FUNCTION_BLOCK FB_IdleState IMPLEMENTS I_State
VAR_INPUT
END_VAR
VAR_OUTPUT
END_VAR
VAR
	pMachine : POINTER TO FB_StateMachine;
END_VAR

{warning 'Eigenschaftenimplementierung hinzufügen'}
PROPERTY Description : STRING
GET
Description := 'Heat pump is idle';
END_GET
END_PROPERTY

METHOD ErrorDetected : BOOL
VAR_INPUT
	errorEvents		: ST_ErrorEvents;
END_VAR
VAR
	message				: STRING(255);
END_VAR
message := toErrorText(errorEvents);
ADSLOGSTR(ADSLOG_MSGTYPE_HINT, 'Error detected -> Error:  %s', message);
pMachine^.SetState(pMachine^.ErrorState);
END_METHOD

//FB_Init ist immer implizit verfügbar und wird primär für die Initialisierung verwendet.
//Der Rückgabewert wird nicht ausgewertet. Für gezielte Einflussnahme können Sie
//die Methoden explizit deklarieren und darin mit dem Standard-Initialisierungscode 
//zusätzlichen Code bereitstellen. Sie können den Rückgabewert auswerten.
METHOD FB_Init: BOOL
VAR_INPUT    
	bInitRetains: BOOL; // TRUE: Die Retain-Variablen werden initialisiert (Reset warm / Reset kalt)    
	bInCopyCode: BOOL;  // TRUE: Die Instanz wird danach in den Kopiercode kopiert (Online-Change)
	pMachine : POINTER TO FB_StateMachine;
END_VAR
THIS^.pMachine := pMachine;
END_METHOD

{warning 'Methodenimplementierung hinzufügen'}
METHOD HeatIsRequested : BOOL
pMachine^.timerTON();

IF pMachine^.timerTON.Q OR NOT pMachine^.timerTON.IN THEN
	ADSLOGSTR(ADSLOG_MSGTYPE_HINT, 'Heizung wurde angefordert -> %s', pMachine^.RunningState.Name);
	pMachine^.timerTON(IN := FALSE);  
	pMachine^.SetState(pMachine^.RunningState);	
END_IF
END_METHOD

{warning 'Methodenimplementierung hinzufügen'}
METHOD LimitValuesAreExceeded : BOOL
END_METHOD

PROPERTY Name : STRING
GET
Name := 'Idle';
END_GET
END_PROPERTY

PROPERTY State : E_State
GET
State := E_State.IDLE;
END_GET
END_PROPERTY

{warning 'Methodenimplementierung hinzufügen'}
METHOD TargetTemeperatureReached : BOOL
END_METHOD

{warning 'Methodenimplementierung hinzufügen'}
METHOD UserPressedConfirmationButton : BOOL
END_METHOD

{warning 'Methodenimplementierung hinzufügen'}
METHOD UserPressedSwitchOffButton : BOOL
END_METHOD

{warning 'Methodenimplementierung hinzufügen'}
METHOD UserPressedSwitchOnButton : BOOL
END_METHOD

{warning 'Methodenimplementierung hinzufügen'}
METHOD WaterHasCooledDown : BOOL
END_METHOD

END_FUNCTION_BLOCK

(* stored: Version 1.1.0.1
   POU FB_IdleState: Id {f7ee3b58-03be-4f49-9ed9-f40543cf4b57}, SpecialFunc None
   Property Description: Id {fe51051b-bde8-49da-adbd-89ef23576803}
   Get Get: Id {448f7325-1a41-4ec7-86c8-2b42eb5aca50}
   Method ErrorDetected: Id {c9936d55-474b-4266-b158-caa16b670de2}
   Method FB_init: Id {b9038d94-a7c9-4cbf-a3fb-ded17a7a84e2}
   Method HeatIsRequested: Id {f9b980c4-904d-441c-b993-50969d377d74}
   Method LimitValuesAreExceeded: Id {14c877c5-3616-4fde-8e7d-07cd27554d4a}
   Property Name: Id {2a551905-1ead-4936-adda-5cd868f31c51}
   Get Get: Id {0cb103a8-6c0b-456d-9502-a94f5cbc533a}
   Property State: Id {3e6615a4-0b72-4744-aa4a-b8431f3a85b9}
   Get Get: Id {cf43e076-33c9-47e4-8b60-ba518cf16a3b}
   Method TargetTemeperatureReached: Id {a8926a6b-0653-4ec9-9337-e0d5d6da7cc7}
   Method UserPressedConfirmationButton: Id {95da523e-2d62-4c12-b016-a3dab2092a78}
   Method UserPressedSwitchOffButton: Id {d42dbbf4-6bf5-457a-84b2-51c8ce6fc5fc}
   Method UserPressedSwitchOnButton: Id {0fd362f1-3f35-42de-86a1-4307d29fa058}
   Method WaterHasCooledDown: Id {0b5f95d5-71c8-41b3-9a09-8b178e27c447} *)
